Universal Robots PolyScope program: junaid_project.urp

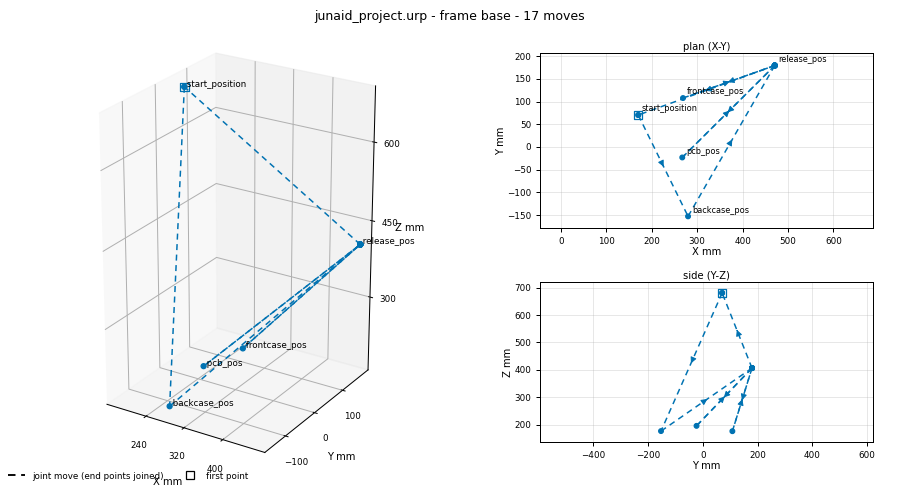
[picture p0: tool path of junaid_project.urp in frame base, 17 of 17 moves have a stored position in this frame; points joined in program order, loops and branches not executed]
Program junaid_project (installation=default directory=/programs/usbdisk/Files createdIn=3.10.0.76181 lastSavedIn=3.10.0.76181 robotSerialNumber=2019330711)
Calibrated DH parameters: a=[0.000088, -0.206409, -0.167255, 0.000029, -0.000053, 0]; d=[0.151895, -39.867408, 110.543254, -70.563598, 0.085358, 0.082453]; alpha=[1.571407, 0.003245, -0.001873, 1.57184, -1.571448, 0]; deltaTheta=[0.000061, -0.559968, -0.109491, 0.66948, 0.000053, -0.000043]
Robot Program (runOnlyOnce=false)
  URCap Gripper Activate (Robotiq_Grippers, Robotiq Inc.) dataModel(ResetAndActivateKey=false)
  Wait Sleep waitTime=10
  URCap Gripper (Robotiq_Grippers, Robotiq Inc.) dataModel(position=0.0, force=25.88235294117647, speed=16.07843137254902, positionInDouble=0.0, forceInDouble=25.88235294117647, speedInDouble=16.07843137254902, slaveIds=[9], blocking=true)
  Loop Counting (count=20) loopVariable(name=Loop_1)
    MoveJ speed 60 deg/s, acceleration 80 deg/s^2 (useActiveTCP=true)
      Waypoint start_position: TCP in base x=170.261 y=70.238 z=680.622 mm, rx=0.1619 ry=1.6568 rz=-0.2375 rad; joints [-195.564, -88.633, 12.108, -98.441, -88.935, 446.443] deg
    MoveJ speed 60 deg/s, acceleration 80 deg/s^2 (useActiveTCP=true)
      Waypoint backcase_pos: TCP in base x=279.896 y=-152.873 z=176.453 mm, rx=0.1471 ry=-3.0634 rz=0.0215 rad; joints [-228.075, -78.52, 115.795, -125.25, -93.964, 396.272] deg
      URCap Gripper (Robotiq_Grippers, Robotiq Inc.) dataModel(position=100.0, force=25.88235294117647, speed=16.07843137254902, positionInDouble=100.0, forceInDouble=25.88235294117647, speedInDouble=16.07843137254902, slaveIds=[9], blocking=true)
      URCap Grip Check (Robotiq_Grippers, Robotiq Inc.) dataModel(ObjectDetectedKey=true, DimensionValidationKey=false, DimensionKey=100.0, DimensionDimensionPositiveGapKey=5.0, DimensionNegativeGapKey=5.0, GripperIdKey=1, ModelDefinedKey=true); state(isChildrenLocked=true)
        URCap If (Robotiq_Grippers, Robotiq Inc.)
          Waypoint release_pos: TCP in base x=470.773 y=179.206 z=406.394 mm, rx=-0.2951 ry=2.3038 rz=0.0698 rad; joints [-172.504, -22.719, -23.715, -90.523, -87.13, 444.106] deg
          URCap Gripper (Robotiq_Grippers, Robotiq Inc.) dataModel(position=0.0, force=16.07843137254902, speed=25.88235294117647, positionInDouble=0.0, forceInDouble=16.07843137254902, speedInDouble=25.88235294117647, slaveIds=[9], blocking=true)
        URCap Else (Robotiq_Grippers, Robotiq Inc.)
          URCap Gripper (Robotiq_Grippers, Robotiq Inc.) dataModel(position=0.0, force=16.07843137254902, speed=25.88235294117647, positionInDouble=0.0, forceInDouble=16.07843137254902, speedInDouble=25.88235294117647, slaveIds=[9], blocking=true)
          URCap Gripper (Robotiq_Grippers, Robotiq Inc.) dataModel(position=100.0, force=16.07843137254902, speed=25.88235294117647, positionInDouble=100.0, forceInDouble=16.07843137254902, speedInDouble=25.88235294117647, slaveIds=[9], blocking=true)
          URCap Grip Check (Robotiq_Grippers, Robotiq Inc.) dataModel(ObjectDetectedKey=true, DimensionValidationKey=false, DimensionKey=100.0, DimensionDimensionPositiveGapKey=5.0, DimensionNegativeGapKey=5.0, GripperIdKey=1, ModelDefinedKey=true); state(isChildrenLocked=true)
            URCap If (Robotiq_Grippers, Robotiq Inc.)
              Waypoint release_pos: TCP in base x=470.773 y=179.206 z=406.394 mm, rx=-0.2951 ry=2.3038 rz=0.0698 rad; joints [-172.504, -22.719, -23.715, -90.523, -87.13, 444.106] deg
              URCap Gripper (Robotiq_Grippers, Robotiq Inc.) dataModel(position=0.0, force=16.07843137254902, speed=25.88235294117647, positionInDouble=0.0, forceInDouble=16.07843137254902, speedInDouble=25.88235294117647, slaveIds=[9], blocking=true)
            URCap Else (Robotiq_Grippers, Robotiq Inc.)
              URCap Gripper (Robotiq_Grippers, Robotiq Inc.) dataModel(position=0.0, force=16.07843137254902, speed=25.88235294117647, positionInDouble=0.0, forceInDouble=16.07843137254902, speedInDouble=25.88235294117647, slaveIds=[9], blocking=true)
              Popup Error (haltProgram=false message=Backcase not detected, please place in first slot inputType=Text)
              URCap Gripper (Robotiq_Grippers, Robotiq Inc.) dataModel(position=100.0, force=16.07843137254902, speed=25.88235294117647, positionInDouble=100.0, forceInDouble=16.07843137254902, speedInDouble=25.88235294117647, slaveIds=[9], blocking=true)
              URCap Grip Check (Robotiq_Grippers, Robotiq Inc.) dataModel(ObjectDetectedKey=true, DimensionValidationKey=false, DimensionKey=100.0, DimensionDimensionPositiveGapKey=5.0, DimensionNegativeGapKey=5.0, GripperIdKey=1, ModelDefinedKey=true); state(isChildrenLocked=true)
                URCap If (Robotiq_Grippers, Robotiq Inc.)
                  Waypoint release_pos: TCP in base x=470.773 y=179.206 z=406.394 mm, rx=-0.2951 ry=2.3038 rz=0.0698 rad; joints [-172.504, -22.719, -23.715, -90.523, -87.13, 444.106] deg
                  URCap Gripper (Robotiq_Grippers, Robotiq Inc.) dataModel(position=0.0, force=16.07843137254902, speed=25.88235294117647, positionInDouble=0.0, forceInDouble=16.07843137254902, speedInDouble=25.88235294117647, slaveIds=[9], blocking=true)
                URCap Else (Robotiq_Grippers, Robotiq Inc.)
                  URCap Gripper (Robotiq_Grippers, Robotiq Inc.) dataModel(position=0.0, force=16.07843137254902, speed=25.88235294117647, positionInDouble=0.0, forceInDouble=16.07843137254902, speedInDouble=25.88235294117647, slaveIds=[9], blocking=true)
                  URCap Gripper (Robotiq_Grippers, Robotiq Inc.) dataModel(position=100.0, force=16.07843137254902, speed=25.88235294117647, positionInDouble=100.0, forceInDouble=16.07843137254902, speedInDouble=25.88235294117647, slaveIds=[9], blocking=true)
                  URCap Grip Check (Robotiq_Grippers, Robotiq Inc.) dataModel(ObjectDetectedKey=true, DimensionValidationKey=false, DimensionKey=100.0, DimensionDimensionPositiveGapKey=5.0, DimensionNegativeGapKey=5.0, GripperIdKey=1, ModelDefinedKey=true); state(isChildrenLocked=true)
                    URCap If (Robotiq_Grippers, Robotiq Inc.)
                      Waypoint release_pos: TCP in base x=470.773 y=179.206 z=406.394 mm, rx=-0.2951 ry=2.3038 rz=0.0698 rad; joints [-172.504, -22.719, -23.715, -90.523, -87.13, 444.106] deg
                      URCap Gripper (Robotiq_Grippers, Robotiq Inc.) dataModel(position=0.0, force=16.07843137254902, speed=25.88235294117647, positionInDouble=0.0, forceInDouble=16.07843137254902, speedInDouble=25.88235294117647, slaveIds=[9], blocking=true)
                    URCap Else (Robotiq_Grippers, Robotiq Inc.)
                      URCap Gripper (Robotiq_Grippers, Robotiq Inc.) dataModel(position=0.0, force=16.07843137254902, speed=25.88235294117647, positionInDouble=0.0, forceInDouble=16.07843137254902, speedInDouble=25.88235294117647, slaveIds=[9], blocking=true)
                      Halt
    MoveJ speed 60 deg/s, acceleration 80 deg/s^2 (useActiveTCP=true)
      Waypoint pcb_pos: TCP in base x=267.16 y=-23.217 z=195.524 mm, rx=0.1564 ry=-3.069 rz=0.0124 rad; joints [-208.77, -93.891, 125.858, -118.911, -92.647, 415.276] deg
      URCap Gripper (Robotiq_Grippers, Robotiq Inc.) dataModel(position=100.0, force=25.88235294117647, speed=16.07843137254902, positionInDouble=100.0, forceInDouble=25.88235294117647, speedInDouble=16.07843137254902, slaveIds=[9], blocking=true)
      URCap Grip Check (Robotiq_Grippers, Robotiq Inc.) dataModel(ObjectDetectedKey=true, DimensionDimensionPositiveGapKey=5.0, DimensionNegativeGapKey=5.0, GripperIdKey=1, ModelDefinedKey=true, DimensionKey=100.0, DimensionValidationKey=false); state(isChildrenLocked=true)
        URCap If (Robotiq_Grippers, Robotiq Inc.)
          Waypoint release_pos: TCP in base x=470.773 y=179.206 z=406.394 mm, rx=-0.2951 ry=2.3038 rz=0.0698 rad; joints [-172.504, -22.719, -23.715, -90.523, -87.13, 444.106] deg
          URCap Gripper (Robotiq_Grippers, Robotiq Inc.) dataModel(position=0.0, force=16.07843137254902, speed=25.88235294117647, positionInDouble=0.0, forceInDouble=16.07843137254902, speedInDouble=25.88235294117647, slaveIds=[9], blocking=true)
        URCap Else (Robotiq_Grippers, Robotiq Inc.)
          URCap Gripper (Robotiq_Grippers, Robotiq Inc.) dataModel(position=0.0, force=16.07843137254902, speed=25.88235294117647, positionInDouble=0.0, forceInDouble=16.07843137254902, speedInDouble=25.88235294117647, slaveIds=[9], blocking=true)
          Popup Error (haltProgram=false message=PCB not detected, please place in second slot inputType=Text)
          URCap Gripper (Robotiq_Grippers, Robotiq Inc.) dataModel(position=100.0, force=16.07843137254902, speed=25.88235294117647, positionInDouble=100.0, forceInDouble=16.07843137254902, speedInDouble=25.88235294117647, slaveIds=[9], blocking=true)
          URCap Grip Check (Robotiq_Grippers, Robotiq Inc.) dataModel(ObjectDetectedKey=true, DimensionValidationKey=false, DimensionKey=100.0, DimensionDimensionPositiveGapKey=5.0, DimensionNegativeGapKey=5.0, GripperIdKey=1, ModelDefinedKey=true); state(isChildrenLocked=true)
            URCap If (Robotiq_Grippers, Robotiq Inc.)
              Waypoint release_pos: TCP in base x=470.773 y=179.206 z=406.394 mm, rx=-0.2951 ry=2.3038 rz=0.0698 rad; joints [-172.504, -22.719, -23.715, -90.523, -87.13, 444.106] deg
              URCap Gripper (Robotiq_Grippers, Robotiq Inc.) dataModel(position=0.0, force=16.07843137254902, speed=25.88235294117647, positionInDouble=0.0, forceInDouble=16.07843137254902, speedInDouble=25.88235294117647, slaveIds=[9], blocking=true)
            URCap Else (Robotiq_Grippers, Robotiq Inc.)
              URCap Gripper (Robotiq_Grippers, Robotiq Inc.) dataModel(position=0.0, force=16.07843137254902, speed=25.88235294117647, positionInDouble=0.0, forceInDouble=16.07843137254902, speedInDouble=25.88235294117647, slaveIds=[9], blocking=true)
              URCap Gripper (Robotiq_Grippers, Robotiq Inc.) dataModel(position=100.0, force=16.07843137254902, speed=25.88235294117647, positionInDouble=100.0, forceInDouble=16.07843137254902, speedInDouble=25.88235294117647, slaveIds=[9], blocking=true)
              URCap Grip Check (Robotiq_Grippers, Robotiq Inc.) dataModel(ObjectDetectedKey=true, DimensionValidationKey=false, DimensionKey=100.0, DimensionDimensionPositiveGapKey=5.0, DimensionNegativeGapKey=5.0, GripperIdKey=1, ModelDefinedKey=true); state(isChildrenLocked=true)
                URCap If (Robotiq_Grippers, Robotiq Inc.)
                  Waypoint release_pos: TCP in base x=470.773 y=179.206 z=406.394 mm, rx=-0.2951 ry=2.3038 rz=0.0698 rad; joints [-172.504, -22.719, -23.715, -90.523, -87.13, 444.106] deg
                  URCap Gripper (Robotiq_Grippers, Robotiq Inc.) dataModel(position=0.0, force=16.07843137254902, speed=25.88235294117647, positionInDouble=0.0, forceInDouble=16.07843137254902, speedInDouble=25.88235294117647, slaveIds=[9], blocking=true)
                URCap Else (Robotiq_Grippers, Robotiq Inc.)
                  URCap Gripper (Robotiq_Grippers, Robotiq Inc.) dataModel(position=0.0, force=16.07843137254902, speed=25.88235294117647, positionInDouble=0.0, forceInDouble=16.07843137254902, speedInDouble=25.88235294117647, slaveIds=[9], blocking=true)
                  URCap Gripper (Robotiq_Grippers, Robotiq Inc.) dataModel(position=100.0, force=16.07843137254902, speed=25.88235294117647, positionInDouble=100.0, forceInDouble=16.07843137254902, speedInDouble=25.88235294117647, slaveIds=[9], blocking=true)
                  URCap Grip Check (Robotiq_Grippers, Robotiq Inc.) dataModel(ObjectDetectedKey=true, DimensionValidationKey=false, DimensionKey=100.0, DimensionDimensionPositiveGapKey=5.0, DimensionNegativeGapKey=5.0, GripperIdKey=1, ModelDefinedKey=true); state(isChildrenLocked=true)
                    URCap If (Robotiq_Grippers, Robotiq Inc.)
                      Waypoint release_pos: TCP in base x=470.773 y=179.206 z=406.394 mm, rx=-0.2951 ry=2.3038 rz=0.0698 rad; joints [-172.504, -22.719, -23.715, -90.523, -87.13, 444.106] deg
                      URCap Gripper (Robotiq_Grippers, Robotiq Inc.) dataModel(position=0.0, force=16.07843137254902, speed=25.88235294117647, positionInDouble=0.0, forceInDouble=16.07843137254902, speedInDouble=25.88235294117647, slaveIds=[9], blocking=true)
                    URCap Else (Robotiq_Grippers, Robotiq Inc.)
                      URCap Gripper (Robotiq_Grippers, Robotiq Inc.) dataModel(position=0.0, force=16.07843137254902, speed=25.88235294117647, positionInDouble=0.0, forceInDouble=16.07843137254902, speedInDouble=25.88235294117647, slaveIds=[9], blocking=true)
                      Halt
    MoveJ speed 60 deg/s, acceleration 80 deg/s^2 (useActiveTCP=true)
      Waypoint frontcase_pos: TCP in base x=268.775 y=107.599 z=176.019 mm, rx=0.1474 ry=-3.0632 rz=0.0217 rad; joints [-180.55, -85.346, 123.071, -123.536, -91.226, 443.773] deg
      URCap Gripper (Robotiq_Grippers, Robotiq Inc.) dataModel(position=100.0, force=16.07843137254902, speed=25.88235294117647, positionInDouble=100.0, forceInDouble=16.07843137254902, speedInDouble=25.88235294117647, slaveIds=[9], blocking=true)
      URCap Grip Check (Robotiq_Grippers, Robotiq Inc.) dataModel(ObjectDetectedKey=true, DimensionValidationKey=false, DimensionKey=100.0, DimensionDimensionPositiveGapKey=5.0, DimensionNegativeGapKey=5.0, GripperIdKey=1, ModelDefinedKey=true); state(isChildrenLocked=true)
        URCap If (Robotiq_Grippers, Robotiq Inc.)
          Waypoint release_pos: TCP in base x=470.773 y=179.206 z=406.394 mm, rx=-0.2951 ry=2.3038 rz=0.0698 rad; joints [-172.504, -22.719, -23.715, -90.523, -87.13, 444.106] deg
          URCap Gripper (Robotiq_Grippers, Robotiq Inc.) dataModel(position=0.0, force=16.07843137254902, speed=25.88235294117647, positionInDouble=0.0, forceInDouble=16.07843137254902, speedInDouble=25.88235294117647, slaveIds=[9], blocking=true)
        URCap Else (Robotiq_Grippers, Robotiq Inc.)
          URCap Gripper (Robotiq_Grippers, Robotiq Inc.) dataModel(position=0.0, force=16.07843137254902, speed=25.88235294117647, positionInDouble=0.0, forceInDouble=16.07843137254902, speedInDouble=25.88235294117647, slaveIds=[9], blocking=true)
          Popup Error (haltProgram=false message=Frontcase not detected, please place in third slot inputType=Text)
          URCap Gripper (Robotiq_Grippers, Robotiq Inc.) dataModel(position=100.0, force=16.07843137254902, speed=25.88235294117647, positionInDouble=100.0, forceInDouble=16.07843137254902, speedInDouble=25.88235294117647, slaveIds=[9], blocking=true)
          URCap Grip Check (Robotiq_Grippers, Robotiq Inc.) dataModel(ObjectDetectedKey=true, DimensionValidationKey=false, DimensionKey=100.0, DimensionDimensionPositiveGapKey=5.0, DimensionNegativeGapKey=5.0, GripperIdKey=1, ModelDefinedKey=true); state(isChildrenLocked=true)
            URCap If (Robotiq_Grippers, Robotiq Inc.)
              Waypoint release_pos: TCP in base x=470.773 y=179.206 z=406.394 mm, rx=-0.2951 ry=2.3038 rz=0.0698 rad; joints [-172.504, -22.719, -23.715, -90.523, -87.13, 444.106] deg
              URCap Gripper (Robotiq_Grippers, Robotiq Inc.) dataModel(position=0.0, force=16.07843137254902, speed=25.88235294117647, positionInDouble=0.0, forceInDouble=16.07843137254902, speedInDouble=25.88235294117647, slaveIds=[9], blocking=true)
            URCap Else (Robotiq_Grippers, Robotiq Inc.)
              URCap Gripper (Robotiq_Grippers, Robotiq Inc.) dataModel(position=0.0, force=16.07843137254902, speed=25.88235294117647, positionInDouble=0.0, forceInDouble=16.07843137254902, speedInDouble=25.88235294117647, slaveIds=[9], blocking=true)
              URCap Gripper (Robotiq_Grippers, Robotiq Inc.) dataModel(position=100.0, force=16.07843137254902, speed=25.88235294117647, positionInDouble=100.0, forceInDouble=16.07843137254902, speedInDouble=25.88235294117647, slaveIds=[9], blocking=true)
              URCap Grip Check (Robotiq_Grippers, Robotiq Inc.) dataModel(ObjectDetectedKey=true, DimensionValidationKey=false, DimensionKey=100.0, DimensionDimensionPositiveGapKey=5.0, DimensionNegativeGapKey=5.0, GripperIdKey=1, ModelDefinedKey=true); state(isChildrenLocked=true)
                URCap If (Robotiq_Grippers, Robotiq Inc.)
                  Waypoint release_pos: TCP in base x=470.773 y=179.206 z=406.394 mm, rx=-0.2951 ry=2.3038 rz=0.0698 rad; joints [-172.504, -22.719, -23.715, -90.523, -87.13, 444.106] deg
                  URCap Gripper (Robotiq_Grippers, Robotiq Inc.) dataModel(position=0.0, force=16.07843137254902, speed=25.88235294117647, positionInDouble=0.0, forceInDouble=16.07843137254902, speedInDouble=25.88235294117647, slaveIds=[9], blocking=true)
                URCap Else (Robotiq_Grippers, Robotiq Inc.)
                  URCap Gripper (Robotiq_Grippers, Robotiq Inc.) dataModel(position=0.0, force=16.07843137254902, speed=25.88235294117647, positionInDouble=0.0, forceInDouble=16.07843137254902, speedInDouble=25.88235294117647, slaveIds=[9], blocking=true)
                  URCap Gripper (Robotiq_Grippers, Robotiq Inc.) dataModel(position=100.0, force=16.07843137254902, speed=25.88235294117647, positionInDouble=100.0, forceInDouble=16.07843137254902, speedInDouble=25.88235294117647, slaveIds=[9], blocking=true)
                  URCap Grip Check (Robotiq_Grippers, Robotiq Inc.) dataModel(ObjectDetectedKey=true, DimensionValidationKey=false, DimensionKey=100.0, DimensionDimensionPositiveGapKey=5.0, DimensionNegativeGapKey=5.0, GripperIdKey=1, ModelDefinedKey=true); state(isChildrenLocked=true)
                    URCap If (Robotiq_Grippers, Robotiq Inc.)
                      Waypoint release_pos: TCP in base x=470.773 y=179.206 z=406.394 mm, rx=-0.2951 ry=2.3038 rz=0.0698 rad; joints [-172.504, -22.719, -23.715, -90.523, -87.13, 444.106] deg
                      URCap Gripper (Robotiq_Grippers, Robotiq Inc.) dataModel(position=0.0, force=16.07843137254902, speed=25.88235294117647, positionInDouble=0.0, forceInDouble=16.07843137254902, speedInDouble=25.88235294117647, slaveIds=[9], blocking=true)
                    URCap Else (Robotiq_Grippers, Robotiq Inc.)
                      URCap Gripper (Robotiq_Grippers, Robotiq Inc.) dataModel(position=0.0, force=16.07843137254902, speed=25.88235294117647, positionInDouble=0.0, forceInDouble=16.07843137254902, speedInDouble=25.88235294117647, slaveIds=[9], blocking=true)
                      Halt
    MoveJ speed 60 deg/s, acceleration 80 deg/s^2 (useActiveTCP=true)
      Waypoint start_position: TCP in base x=170.261 y=70.238 z=680.622 mm, rx=0.1619 ry=1.6568 rz=-0.2375 rad; joints [-195.564, -88.633, 12.108, -98.441, -88.935, 446.443] deg
    Wait Sleep waitTime=10
